	{attribute 'OPC.UA.DA' := '1'}  				                
	SP_adsorb_during_steam_bypass										: BOOL;	
	{attribute 'OPC.UA.DA' := '1'}  				                
	SP_adsorb_during_warmup												: BOOL;
	{attribute 'OPC.UA.DA' := '1'}  				                
	SP_boiler_warmup_duration											: REAL;
	{attribute 'OPC.UA.DA' := '1'}  				                
	SP_condensate_collection_tank_high_level							: REAL;	
	{attribute 'OPC.UA.DA' := '1'}  				                
	SP_condensate_collection_tank_low_level								: REAL;
	{attribute 'OPC.UA.DA' := '1'}  				                
	SP_condensation_collection_tank_emergency_low_level					: REAL;	
	{attribute 'OPC.UA.DA' := '1'}  				                
	SP_duration_to_drain_cooling_and_purge_line_in_module				: REAL;				
	{attribute 'OPC.UA.DA' := '1'}  				                
	SP_duration_to_drain_reactor_set									: REAL;	
	{attribute 'OPC.UA.DA' := '1'}  				                
	SP_evacuation_duration												: REAL;							// PS 11/25/24	
	{attribute 'OPC.UA.DA' := '1'}  				                
	SP_evacuation_ideal_pressure										: REAL;							// PS 11/25/24	
	{attribute 'OPC.UA.DA' := '1'}  				                
	SP_mass_flow_totalizer												: REAL;
	{attribute 'OPC.UA.DA' := '1'}  				                
	SP_maximum_condensate_collection_tank_refill_duration				: REAL;							// PS 08_16_24
	{attribute 'OPC.UA.DA' := '1'}  				                
	SP_maximum_condenser_knockout_drain_duration						: REAL;							// PS 08_22_24
	{attribute 'OPC.UA.DA' := '1'}  				                
	SP_maximum_duration_to_drain_reactor_set							: REAL;	
	{attribute 'OPC.UA.DA' := '1'}  				                
	SP_maximum_inlet_product_vacuum_temperature							: REAL;							// PS 04_30_24	
	{attribute 'OPC.UA.DA' := '1'}  				                
	SP_maximum_reasonable_sorbent_TC_reading							: REAL;
	{attribute 'OPC.UA.DA' := '1'}  				                
	SP_maximum_vacuum_separator_drain_duration							: REAL;							// PS 08_22_24
	{attribute 'OPC.UA.DA' := '1'}  				                
	SP_maximum_vacuum_separator_refill_duration							: REAL;							// PS 08_22_24
	{attribute 'OPC.UA.DA' := '1'}  				                
	SP_minimum_condensate_flow											: REAL;							// PS 08_22_24
	{attribute 'OPC.UA.DA' := '1'}  				                
	SP_minimum_dead_air_line_pressure									: REAL;							// PS 11/27/24
	{attribute 'OPC.UA.DA' := '1'}  				                
	SP_minimum_drainage_pressure										: REAL;	
	{attribute 'OPC.UA.DA' := '1'}  				                
	SP_minimum_reasonable_sorbent_TC_reading							: REAL;
	{attribute 'OPC.UA.DA' := '1'}  				                
	SP_minimum_steam_bypass_duration									: REAL;							// PS 12/2/24
	{attribute 'OPC.UA.DA' := '1'}  				                
	SP_minimum_steam_bypass_flow_rate									: REAL;
	{attribute 'OPC.UA.DA' := '1'}  				                
	SP_minimum_vacuum_cooling_loop_flow									: REAL := 2; 						// PS 11/25/24
	{attribute 'OPC.UA.DA' := '1'}  				                
	SP_max_vacuum_cooling_loop_temp										: REAL := 50;							// PS 11/25/24
	{attribute 'OPC.UA.DA' := '1'}  				                
	SP_minimum_vacuum_liq_seal_flow										: REAL;							// PS 08_13_24
	{attribute 'OPC.UA.DA' := '1'}  				                
	SP_product_condensate_drum_high_level								: REAL;
	{attribute 'OPC.UA.DA' := '1'}  				                
	SP_product_condensate_drum_low_level								: REAL;
	{attribute 'OPC.UA.DA' := '1'}  				                
	SP_reactor_vfd_percent_maximum										: INT;
	{attribute 'OPC.UA.DA' := '1'}  				                
	SP_reactor_vfd_percent_step_duration								: REAL;
	{attribute 'OPC.UA.DA' := '1'}  				                
	SP_reactor_vfd_percent_step_size									: INT;
	{attribute 'OPC.UA.DA' := '1'}  				                
	SP_steam_bypass_duration											: REAL;
	{attribute 'OPC.UA.DA' := '1'}  				                
	SP_steam_bypass_immediately_after_warm_up							: BOOL;
	{attribute 'OPC.UA.DA' := '1'}  				                
	SP_steam_bypass_temperature											: REAL;
	{attribute 'OPC.UA.DA' := '1'}  				                
	SP_steam_bypass_vacuum_pressure										: REAL;
	{attribute 'OPC.UA.DA' := '1'}  				                
	SP_target_boiler_pressure											: REAL;
	{attribute 'OPC.UA.DA' := '1'}  				                
	SP_vacuum_pres_control_valve										: REAL;
	{attribute 'OPC.UA.DA' := '1'}  				                
	SP_vacuum_separator_level_emergency_high							: REAL;							// PS 08_13_24									
	{attribute 'OPC.UA.DA' := '1'}  				                
	SP_vacuum_separator_level_emergency_low								: REAL;							// PS 08_13_24									
	{attribute 'OPC.UA.DA' := '1'}  				                
	SP_vacuum_separator_level_high										: REAL;							// PS 08_22_24									
	{attribute 'OPC.UA.DA' := '1'}  				                
	SP_vacuum_separator_level_mid										: REAL;							// PS 08_22_24									
	{attribute 'OPC.UA.DA' := '1'}  				                
	SP_vacuum_separator_level_low										: REAL;							// PS 08_22_24	
	{attribute 'OPC.UA.DA' := '1'}  				                
	SP_waste_water_tank_weight_full										: REAL;										
	{attribute 'OPC.UA.DA' := '1'}  				                
	SP_waste_water_tank_weight_empty									: REAL;	
	{attribute 'OPC.UA.DA' := '1'}  				                
	SP_steam_water_tank_weight_full										: REAL;										
	{attribute 'OPC.UA.DA' := '1'}  				                
	SP_steam_water_tank_weight_empty									: REAL;	
	
	
	
    /// <summary>PCV01</summary>
	vacuum_pres_control_valve_setpoint									: REAL;
	
END_VAR

// Theseus - P_U01
// Rev 1.0 - December 2, 2024

A_IO_Points();
A_PIDs();
A_MovingAverage();
A02_WarmUp();
A03_Steam_Bypass();
A08_Shutdown();
A09_Pressure_Drop_Test();
P_U01.shutdown_process													:= FALSE;

IF LEFT(gsCycleMode, 1) = '0' THEN
	IF gsCycleMode = '02' THEN
		i2Step															:= 1;
	ELSIF gsCycleMode = '03' THEN
		i3Step															:= 1;
	ELSIF gsCycleMode = '08' THEN
		i8Step															:= 1;
	ELSIF gsCycleMode = '09' THEN
		i9Step															:= 1;
	END_IF
	gsCycleMode															:= '';
END_IF

IF tonWriteData.Q OR P_U01.write_persistent_data THEN
	P_U01.write_persistent_data											:= FALSE;
	bWriteData															:= TRUE;
ELSIF NOT fbWriteData.BUSY THEN
	bWriteData															:= FALSE;
END_IF

fbWriteData(	NETID													:= '',
				PORT													:= 851,
				START													:= bWriteData,
				TMOUT													:= T#5S);

tonTimer(IN:= bTimer, PT:= REAL_TO_TIME(rTime));
tonAdsorptionTimer(IN:= bAdsorptionTimer, PT:= REAL_TO_TIME(P_M01.SP_adsorption_duration * _MINUTES));
tonWriteData(IN:= NOT bWriteData, PT:= T#30M);

// Water Scales
fb_WaterScales_In ( 
			i_value := water_scale_1 + water_scale_2,
			io_reset	:= water_scales_reset,
			o_change_value => water_scales_in_delta,
			o_change_rate => water_scales_in_rate
			);
			
fb_WaterScales_Out ( 
			i_value := water_scale_3,
			io_reset	:= water_scales_reset,
			o_change_value => water_scales_out_delta,
			o_change_rate => water_scales_out_rate
			);
		
IF water_scales_reset THEN
	water_scales_reset := FALSE;
END_IF

// Water Scales Capapcity Desorption 
condenser_tank_capacity := SP_waste_water_tank_weight_full - SP_waste_water_tank_weight_empty;
steam_delivery_tank_capacity := SP_steam_water_tank_weight_full - SP_steam_water_tank_weight_empty;
condenser_tank_room_before_full	:= SP_waste_water_tank_weight_full - water_scale_3;
steam_delivery_tank_before_empty := (water_scale_1 + water_scale_2) -  SP_steam_water_tank_weight_empty;

ACTION A_IO_Points:
// Theseus - A_IO_Points
// Rev 1.0 - November 26, 2024

interlock_condenser_steam_or_status										:= interlock_condenser_steam_or;
interlock_hot_reactor_condenser_or_status								:= interlock_hot_reactor_condenser_or;
interlock_no_steam_unevacuated_reactor_or_status						:= interlock_no_steam_unevacuated_reactor_or;
interlock_cooling_with_vacuum_or_status									:= interlock_cooling_with_vacuum_or;
interlock_separator_water_level_with_vacuum_or_status					:= interlock_separator_water_level_with_vacuum_or;
interlock_cooling_loop_flow_with_vacuum_or_status						:= interlock_cooling_loop_flow_with_vacuum_or;
interlock_condensate_tank_level_for_steam_or_status						:= interlock_condensate_tank_level_for_steam_or;
interlock_hot_sorbent_for_repressurization_or_status					:= interlock_hot_sorbent_for_repressurization_or;
interlock_reactor_over_safe_pressure_limit_or_status					:= interlock_reactor_over_safe_pressure_limit_or;
interlock_reactor_over_safe_temperature_limit_or_status					:= interlock_reactor_over_safe_temperature_limit_or;
interlock_repressurization_valve_with_steam_or_status					:= interlock_repressurization_valve_with_steam_or;
interlock_door_open_with_steam_flow_or_status							:= interlock_door_open_with_steam_flow_or;
interlock_door_open_with_reactor_vacuum_or_status						:= interlock_door_open_with_reactor_vacuum_or;
interlock_co2_adsorption_or_status										:= interlock_co2_adsorption_or;
interlock_condensate_pump_or_status										:= interlock_condensate_pump_or;
condenser_knockout_drain_or_on_status									:= condenser_knockout_drain_or_on;
condenser_knockout_drain_or_off_status									:= condenser_knockout_drain_or_off;
vacuum_separator_drain_or_on_status										:= vacuum_separator_drain_or_on;
vacuum_separator_drain_or_off_status									:= vacuum_separator_drain_or_off;
reactor_drain_or_on_status												:= reactor_drain_or_on;
reactor_drain_or_off_status												:= reactor_drain_or_off;

// Interlock 5
cooling_with_vacuum_interlock											:= NOT vacuum_liquid_loop_fan OR NOT vacuum_liquid_pump;
bCondition1																:= NOT interlock_cooling_with_vacuum_or AND cooling_with_vacuum_interlock;

// Interlock 6
separator_water_level_with_vacuum_interlock								:= vacuum_separator_level < SP_vacuum_separator_level_emergency_low OR vacuum_separator_level > SP_vacuum_separator_level_emergency_high;
bCondition2																:= NOT interlock_separator_water_level_with_vacuum_or AND separator_water_level_with_vacuum_interlock;

// Interlock 7
cooling_loop_flow_with_vacuum_interlock									:= vacuum_pump AND vacuum_pump_water_flow < SP_minimum_vacuum_liq_seal_flow;
tonVacuumInterlock(IN:= cooling_loop_flow_with_vacuum_interlock, PT:= T#5S);
bCondition3																:= NOT interlock_cooling_loop_flow_with_vacuum_or AND tonVacuumInterlock.Q;

IF bCondition1 OR bCondition2 OR bCondition3 THEN
	vacuum_pump															:= FALSE;
END_IF
IF bCondition2 THEN
	vacuum_pump_inlet_valve												:= FALSE;
	vacuum_pump_bypass_valve											:= FALSE;
	dead_air_inlet_valve												:= FALSE;
	product_line_ambient_valve											:= INT_TO_BOOL(eAmbient);
END_IF

// Interlock 8
condensate_tank_level_for_steam_interlock								:= steam_water_tank_level < SP_condensation_collection_tank_emergency_low_level;
IF NOT interlock_condensate_tank_level_for_steam_or AND condensate_tank_level_for_steam_interlock THEN
	boiler_package														:= FALSE;
	steam_water_pump													:= FALSE;
	steam_flow_control_valve											:= _CLOSED;
END_IF

gbDrainageOn															:= (drainage_on AND NOT drainage_function_off_or) OR drainage_function_on_or;

// Interlock 9
hot_sorbent_for_repressurization_interlock								:= P_M01.rs1.sorbent_high_temp >= P_M01.SP_maximum_target_sorbent_temperature_to_repressurize;
bCondition1																:= NOT interlock_hot_sorbent_for_repressurization_or AND hot_sorbent_for_repressurization_interlock;
 
// Interlock 13
P_U01.repressurization_valve_with_steam_interlock						:= NOT P_U01.steam_flow_control_valve_closed;
bCondition2																:= NOT P_U01.interlock_repressurization_valve_with_steam_or AND P_U01.repressurization_valve_with_steam_interlock;

gbRepresValves															:= NOT bCondition1 AND NOT bCondition2;

// Vacuum Separator
IF (gbDrainageOn OR vacuum_separator_drain_or_on) AND NOT vacuum_separator_drain_or_off THEN
	// Fill
	tonVacuumSeparatorFill(IN:= tap_water_feed_valve AND NOT bVacuumSeparatorFillError, PT:= REAL_TO_TIME(SP_maximum_vacuum_separator_refill_duration * _MINUTES));
	IF tonVacuumSeparatorFill.Q THEN
		tap_water_feed_valve											:= FALSE;
		bVacuumSeparatorFillError										:= TRUE;
		P_Alarms.M_Add_Alarm(_U01, gsVacuumSeparatorFillError, gsMessageTBD);
	ELSIF vacuum_separator_level < SP_vacuum_separator_level_low  AND NOT bVacuumSeparatorFillError THEN
		tap_water_feed_valve											:= TRUE;
	ELSIF vacuum_separator_level > SP_vacuum_separator_level_mid THEN
		tap_water_feed_valve											:= FALSE;
		bVacuumSeparatorFillError										:= FALSE;
	END_IF
	// Drain
//	tonVacuumSeparatorDrain(IN:= separator_drain_valve AND NOT bVacuumSeparatorDrainError, PT:= REAL_TO_TIME(SP_maximum_vacuum_separator_drain_duration * _MINUTES));
	IF tonVacuumSeparatorFill.Q THEN
		separator_drain_valve											:= FALSE;
		vacuum_separator_drain_pump										:= FALSE;
		bVacuumSeparatorDrainError										:= TRUE;
		P_Alarms.M_Add_Alarm(_U01, gsVacuumSeparatorDrainError, gsMessageTBD);
	ELSIF vacuum_separator_level >= SP_vacuum_separator_level_high THEN
		separator_drain_valve											:= TRUE;
		vacuum_separator_drain_pump										:= TRUE;
	ELSIF vacuum_separator_level < SP_vacuum_separator_level_mid THEN
		separator_drain_valve											:= FALSE;
		vacuum_separator_drain_pump										:= FALSE;
		bVacuumSeparatorDrainError										:= FALSE;
	END_IF
END_IF
rtrigVacuumSeparator(CLK:= NOT gbDrainageOn AND NOT vacuum_separator_drain_or_on AND NOT vacuum_separator_drain_or_off);
IF rtrigVacuumSeparator.Q THEN
	tap_water_feed_valve												:= FALSE;
	separator_drain_valve												:= FALSE;
	vacuum_separator_drain_pump											:= FALSE;
END_IF

// Condenser Knockout drainage
IF (gbDrainageOn OR condenser_knockout_drain_or_on) AND NOT condenser_knockout_drain_or_off THEN
	IF gbCondenserKODrainageOn THEN
//		tonCondenserKODrain(IN:= NOT bCondenserKnockoutError AND (product_condensate_drum_lsh OR product_condensate_drum_lsl), PT:= REAL_TO_TIME(SP_maximum_condenser_knockout_drain_duration * _MINUTES));
		IF tonCondenserKODrain.Q AND P_M01.rs1.reactor_condensate_flow < SP_minimum_condensate_flow THEN
			bCondenserKnockoutError										:= TRUE;
			knockout_drain_valve										:= FALSE;
			steam_flow_control_valve									:= _CLOSED;
			P_Alarms.M_Add_Alarm(_U01, gsCondenserKODrainageError, gsMessageTBD);
		ELSIF product_condensate_drum_lsh THEN
			knockout_drain_valve										:= TRUE;
		ELSIF NOT product_condensate_drum_lsh AND NOT product_condensate_drum_lsl THEN
			knockout_drain_valve										:= FALSE;
		END_IF
	ELSE
		knockout_drain_valve											:= FALSE;
	END_IF
END_IF
rtrigKODrainValve(CLK:= NOT gbDrainageOn AND NOT condenser_knockout_drain_or_on AND NOT condenser_knockout_drain_or_off);
IF rtrigKODrainValve.Q THEN
	knockout_drain_valve												:= FALSE;
END_IF

fb_adsorp_product_wastewater
	( i_execute := condenser_knockout_drain_adsorption_on,
	  i_value := P_U01.water_scale_3,
	  i_time := 30,
	  i_threshold := 1);
	  
IF condenser_knockout_drain_adsorption_on THEN
	IF NOT fb_adsorp_product_wastewater.o_below_threshold THEN
		knockout_drain_valve											:= TRUE;
	ELSIF fb_adsorp_product_wastewater.o_below_threshold OR fb_adsorp_product_wastewater.o_timeout THEN
		knockout_drain_valve											:= FALSE;
		condenser_knockout_drain_adsorption_on 							:= FALSE;
	END_IF
END_IF


IF NOT interlock_condensate_pump_or THEN
	condensate_pump														:= knockout_drain_valve OR gbCondensateValve;
END_IF

// Interlock 2
condenser_steam_interlock												:= NOT steam_flow_control_valve_closed AND (P_M01.rs1.steam_bypass_valve_open OR P_M01.rs1.product_iso_valve_open);
IF NOT interlock_condenser_steam_or AND condenser_steam_interlock THEN
	condenser_pump														:= TRUE;
	condenser_fan														:= TRUE;
END_IF

B_01																	:= boiler_package;
boiler_package_cmd_status												:= B_01;

P_01																	:= steam_water_pump;
steam_water_pump_cmd_status												:= P_01;

P_02																	:= vacuum_pump;
vacuum_pump_cmd_status													:= P_02;

P_03																	:= condensate_pump;
condensate_pump_cmd_status												:= P_03;

P_04																	:= condenser_pump;
condenser_pump_cmd_status												:= P_04;

P_05																	:= vacuum_liquid_pump;
vacuum_liquid_pump_cmd_status											:= P_05;

P_06																	:= vacuum_separator_drain_pump;
vacuum_separator_drain_pump_cmd_status									:= P_06;

E_01																	:= condenser_fan;
condenser_fan_cmd_status												:= E_01; 

X_01																	:= vacuum_liquid_loop_fan;
vacuum_liquid_loop_fan_cmd_status										:= X_01;

product_outlet_co2														:= F_AnalogIn(AT_02, product_outlet_co2_low, product_outlet_co2_high, product_outlet_co2_min, product_outlet_co2_offset);
product_outlet_co2_error												:= AT_02_error AND NOT _ProductOutletCO2ErrorOff;
bProductOutletCo2Error													:= P_Alarms.M_Check_Error(product_outlet_co2_error, bProductOutletCo2Error, _U01, gsProductOutletCo2SensorError, gsProcessCannotRun);

product_outlet_h2o														:= F_AnalogIn(AT_03, product_outlet_h2o_low, product_outlet_h2o_high, product_outlet_h2o_min, product_outlet_h2o_offset);
product_outlet_h2o_error												:= AT_03_error AND NOT _ProductOutletH2OErrorOff;
bProductOutletH2oError													:= P_Alarms.M_Check_Error(product_outlet_h2o_error, bProductOutletH2oError, _U01, gsProductOutletH2oSensorError, gsProcessCannotRun);

product_outlet_flow														:= F_AnalogIn(FT_02, product_outlet_flow_low, product_outlet_flow_high, product_outlet_flow_min, product_outlet_flow_offset);
product_outlet_flow_error												:= product_outlet_flow_error AND NOT _ProductOutletFlowErrorOff;
bProductOutletFlowError													:= P_Alarms.M_Check_Error(product_outlet_flow_error, bProductOutletFlowError, _U01, gsProductOutletFlowSensorError, gsProcessCannotRun);

condensate_flow															:= F_AnalogIn(FT_04, condensate_flow_low, condensate_flow_high, condensate_flow_min, condensate_flow_offset);
condensate_flow_error													:= FT_04_error AND NOT _CondensateFlowErrorOff;
bCondensateFlowError													:= P_Alarms.M_Check_Error(condensate_flow_error, bCondensateFlowError, _U01, gsCondensateFlowSensorError, gsProcessCannotRun);
	
tap_water_feed_flow														:= F_AnalogIn(FT_05, tap_water_feed_flow_low, tap_water_feed_flow_high, tap_water_feed_flow_min, tap_water_feed_flow_offset);
tap_water_feed_flow_error												:= FT_05_error AND NOT _TapWaterFeedFlowErrorOff;
bWaterFeedFlowError														:= P_Alarms.M_Check_Error(tap_water_feed_flow_error, bWaterFeedFlowError, _U01, gsTapWaterFeedFlowSensorError, gsProcessCannotRun);

steam_flow																:= F_AnalogIn(FT_06, steam_flow_low, steam_flow_high, steam_flow_min, steam_flow_offset);
steam_flow_error														:= FT_06_error AND NOT _SteamFlowErrorOff;
bSteamFlowError															:= P_Alarms.M_Check_Error(steam_flow_error, bSteamFlowError, _U01, gsTapWaterFeedFlowSensorError, gsProcessCannotRun);

vacuum_pump_water_flow													:= F_AnalogIn(FT_07, vacuum_pump_water_flow_low, vacuum_pump_water_flow_high, vacuum_pump_water_flow_min, vacuum_pump_water_flow_offset);
vacuum_pump_water_flow_error											:= FT_07_error AND NOT _VacuumPumpWaterFlowErrorOff;
bVacuumPumpWaterFlowError												:= P_Alarms.M_Check_Error(vacuum_pump_water_flow_error, bVacuumPumpWaterFlowError, _U01, gsVacuumPumpWaterFlowSensorError, gsProcessCannotRun);
	
condenser_flow															:= F_AnalogIn(FT_08, condenser_flow_low, condenser_flow_high, condenser_flow_min, condenser_flow_offset);
condenser_flow_error													:= FT_08_error AND NOT _CondenserFlowErrorOff;
bCondenserFlowError														:= P_Alarms.M_Check_Error(condenser_flow_error, bCondenserFlowError, _U01, gsCondenserFlowSensorError, gsProcessCannotRun);
	
steam_water_tank_level													:= F_AnalogIn(LT_01, steam_water_tank_level_low, steam_water_tank_level_high, steam_water_tank_level_min, steam_water_tank_level_offset);
steam_water_tank_level_error											:= LT_01_error AND NOT _SteamWaterTankLevelErrorOff;
bSteamWaterTankLevelError												:= P_Alarms.M_Check_Error(steam_water_tank_level_error, bSteamWaterTankLevelError, _U01, gsSteamWaterTankLevelSensorError, gsProcessCannotRun);
	
vacuum_separator_level													:= F_AnalogIn(LT_02, vacuum_separator_level_low, vacuum_separator_level_high, vacuum_separator_level_min, vacuum_separator_level_offset);
vacuum_separator_level_error											:= LT_02_error AND NOT _VacuumSeparatorLevelErrorOff;
bVacuumSeparatorLevelError												:= P_Alarms.M_Check_Error(vacuum_separator_level_error, bVacuumSeparatorLevelError, _U01, gsVacuumSeparatorLevelSensorError, gsProcessCannotRun);
	
product_vacuum_pres														:= F_AnalogIn(PT_04, product_vacuum_pres_low, product_vacuum_pres_high, product_vacuum_pres_min, product_vacuum_pres_offset);
product_vacuum_pres_error												:= PT_04_error AND NOT _ProductVacuumPresErrorOff;
bProductVacuumPresError													:= P_Alarms.M_Check_Error(product_vacuum_pres_error, bProductVacuumPresError, _U01, gsProductVacuumPresSensorError, gsProcessCannotRun);

steam_line_pres															:= F_AnalogIn(PT_07, steam_line_pres_low, steam_line_pres_high, steam_line_pres_min, steam_line_pres_offset);
steam_line_pres_error													:= PT_07_error AND NOT _SteamLinePresErrorOff;
bSteamLinePresError														:= P_Alarms.M_Check_Error(steam_line_pres_error, bSteamLinePresError, _U01, gsSteamLinePresSensorError, gsProcessCannotRun);

flow_calibration_diff_pres												:= F_AnalogIn(PDT_04, flow_calibration_diff_pres_low, flow_calibration_diff_pres_high, flow_calibration_diff_pres_min, flow_calibration_diff_pres_offset);
flow_calibration_diff_pres_error										:= PDT_04_error AND NOT _FlowCalibrationDiffPresErrorOff;
bFlowCalibrationDiffPresError											:= P_Alarms.M_Check_Error(flow_calibration_diff_pres_error, bFlowCalibrationDiffPresError, _U01, gsFlowCalibrationDiffPresSensorError, gsProcessCannotRun);


water_scale_1															:= F_AnalogIn(WI_01, water_scale_1_low, water_scale_1_high, water_scale_1_min, water_scale_1_offset);
water_scale_1_error														:= WI_01_error AND NOT _WaterScale1ErrorOff;
bWaterScale1Error														:= P_Alarms.M_Check_Error(water_scale_1_error, bWaterScale1Error, _U01, gsWaterScale1SensorError, gsWarning); 
	
water_scale_2															:= F_AnalogIn(WI_02, water_scale_2_low, water_scale_2_high, water_scale_2_min, water_scale_2_offset);
water_scale_2_error														:= WI_02_error AND NOT _WaterScale2ErrorOff;
bWaterScale2Error														:= P_Alarms.M_Check_Error(water_scale_2_error, bWaterScale2Error, _U01, gsWaterScale1SensorError, gsWarning); 

water_scale_3															:= F_AnalogIn(WI_03, water_scale_3_low, water_scale_3_high, water_scale_3_min, water_scale_3_offset);
water_scale_3_error														:= WI_03_error AND NOT _WaterScale3ErrorOff;
bWaterScale3Error														:= P_Alarms.M_Check_Error(water_scale_3_error, bWaterScale3Error, _U01, gsWaterScale1SensorError, gsWarning);

product_temp															:= F_Temperature(TT_02, product_temp_offset);
product_temp_error														:= TT_02_error AND NOT _ProductTempErrorOff;
bProductTempError														:= P_Alarms.M_Check_Error(product_temp_error, bProductTempError, _U01, gsProductTempSensorError, gsProcessCannotRun);

product_vacuum_temp														:= F_Temperature(TT_03, product_vacuum_temp_offset);
product_vacuum_temp_error												:= TT_03_error AND NOT _ProductVacuumTempOff;
bProductVacuumTempError													:= P_Alarms.M_Check_Error(product_vacuum_temp_error, bProductVacuumTempError, _U01, gsProductVacuumTempSensorError, gsProcessCannotRun);
	
inlet_line_temp															:= F_Temperature(TT_06, inlet_line_temp_offset);
inlet_line_temp_error													:= TT_06_error AND NOT _InletLineTempErrorOff;
bInletLineTempError														:= P_Alarms.M_Check_Error(inlet_line_temp_error, bInletLineTempError, _U01, gsInletLineTempSensorError, gsProcessCannotRun);

vacuum_pump_water_temp_1												:= F_Temperature(TT_10, vacuum_pump_water_temp_1_offset);
vacuum_pump_water_temp_1_error											:= TT_10_error AND NOT _VacuumPumpWaterTemp1ErrorOff;
bVacuumPumpWaterTemp1Error												:= P_Alarms.M_Check_Error(vacuum_pump_water_temp_1_error, bVacuumPumpWaterTemp1Error, _U01, gsVacuumPumpWaterTemp1SensorError, gsProcessCannotRun);

vacuum_pump_water_temp_2												:= F_Temperature(TT_11, vacuum_pump_water_temp_2_offset);
vacuum_pump_water_temp_2_error											:= TT_11_error AND NOT _VacuumPumpWaterTemp2ErrorOff;

IF bCloseXVValves THEN
	vacuum_pump_inlet_valve												:= FALSE;
	vacuum_pump_bypass_valve											:= FALSE;
	knockout_drain_valve												:= FALSE;
	dead_air_inlet_valve												:= FALSE;
	separator_drain_valve												:= FALSE;
	bCloseXVValves														:= FALSE;
END_IF

XV_03																	:= 	vacuum_pump_inlet_valve;
vacuum_pump_inlet_valve_open_cmd_status									:= vacuum_pump_inlet_valve;
vacuum_pump_inlet_valve_clear											:= F_ValveClear(vacuum_pump_inlet_valve, vacuum_pump_inlet_valve_open, vacuum_pump_inlet_valve_closed);

XV_04																	:= vacuum_pump_bypass_valve;
vacuum_pump_bypass_valve_open_cmd_status								:= XV_04;
vacuum_pump_bypass_valve_clear											:= F_ValveClear(vacuum_pump_bypass_valve, vacuum_pump_bypass_valve_open, vacuum_pump_bypass_valve_closed);

XV_06																	:= knockout_drain_valve;
knockout_drain_valve_open_cmd_status									:= XV_06;
knockout_drain_valve_clear												:= F_ValveClear(knockout_drain_valve, knockout_drain_valve_open, knockout_drain_valve_closed);

XV_10																	:= dead_air_inlet_valve;
dead_air_inlet_valve_open_cmd_status									:= dead_air_inlet_valve;
dead_air_inlet_valve_clear												:= F_ValveClear(dead_air_inlet_valve, dead_air_inlet_valve_open, dead_air_inlet_valve_closed);

XV_11																	:= product_line_ambient_valve;
product_line_ambient_valve_cmd_status									:= XV_11;
product_line_ambient_valve_clear										:= F_ValveClear(product_line_ambient_valve, product_line_ambient_valve_ambient,product_line_ambient_valve_product);

XV_12																	:= tap_water_feed_valve;
tap_water_feed_valve_cmd_status											:= XV_12;

XV_13																	:= separator_drain_valve;
separator_drain_valve_open_cmd_status									:= XV_13;
separator_drain_valve_clear												:= F_ValveClear(separator_drain_valve, separator_drain_valve_open, separator_drain_valve_closed);

XV_14																	:= steam_water_reservoir_valve;
steam_water_reservoir_valve_cmd_status									:= XV_14;

fb_Vacuum_Pres_Control_Valve_PI(		Setpoint						:= vacuum_pres_control_valve_setpoint,
										Control							:= product_vacuum_pres,
										Error							:= vacuum_pres_control_valve_position_error,
										Reverse							:= FALSE,
										Kp								:= vacuum_pres_control_valve_kp,           
										Ki								:= vacuum_pres_control_valve_ki,           
										BaseAdjust						:= vacuum_pres_control_valve_base_adjust,  
										LoopTime						:= vacuum_pres_control_valve_loop_time,    
										IBand							:= vacuum_pres_control_valve_iband,        
										Base							:= vacuum_pres_control_valve_base,         
										Mode							:= vacuum_pres_control_valve_mode,
										Input							:= vacuum_pres_control_valve,
										Mode_Out						=> vacuum_pres_control_valve_current_mode, 
										Output							=> PCV_01);

vacuum_pres_control_valve_position										:= INT_TO_REAL(PCV_01_position) / _PERCENT_FACTOR; 
vacuum_pres_control_valve_open											:= vacuum_pres_control_valve_position >= _VALVE_OPEN;
vacuum_pres_control_valve_closed										:= vacuum_pres_control_valve_position < _VALVE_CLOSED;

fb_Steam_Flow_Control_Valve_PI(			Setpoint						:= steam_flow_control_valve_setpoint,
										Control							:= ,
										Error							:= steam_flow_control_valve_position_error,
										Reverse							:= FALSE,
										Kp								:= steam_flow_control_valve_kp,           
										Ki								:= steam_flow_control_valve_ki,           
										BaseAdjust						:= steam_flow_control_valve_base_adjust,  
										LoopTime						:= steam_flow_control_valve_loop_time,    
										IBand							:= steam_flow_control_valve_iband,        
										Base							:= steam_flow_control_valve_base,         
										Mode							:= steam_flow_control_valve_mode,
										Input							:= steam_flow_control_valve,
										Mode_Out						=> steam_flow_control_valve_current_mode, 
										Output							=> PCV_02);

steam_flow_control_valve_position										:= INT_TO_REAL(PCV_02_position) / _PERCENT_FACTOR; 
steam_flow_control_valve_open											:= steam_flow_control_valve_position >= _VALVE_OPEN;
steam_flow_control_valve_closed											:= steam_flow_control_valve_position < _VALVE_CLOSED;

// ignore if < 2 Amps
l1_current_240															:= SEL(IT1 > _CURRENT_240_FACTOR * 2,0,F_IEConvert(IT1, _CURRENT_240_FACTOR));
l2_current_240															:= SEL(IT2 > _CURRENT_240_FACTOR * 2,0,F_IEConvert(IT2, _CURRENT_240_FACTOR));
l3_current_240															:= SEL(IT3 > _CURRENT_240_FACTOR * 2,0,F_IEConvert(IT3, _CURRENT_240_FACTOR));
l1_voltage_240															:= F_IEConvert(VT1, _VOLTAGE_240_FACTOR);
l2_voltage_240															:= F_IEConvert(VT2, _VOLTAGE_240_FACTOR);
l3_voltage_240															:= F_IEConvert(VT3, _VOLTAGE_240_FACTOR);

// Ignore if < 1 Amp
l1_current_120															:= SEL(IT4 > _CURRENT_120_FACTOR ,0,F_IEConvert(IT4, _CURRENT_120_FACTOR));
l1_voltage_120															:= F_IEConvert(VT4, _VOLTAGE_120_FACTOR);

// Boiler - ignore noise if < 5A = 400 counts

l1_current_boiler := SEL(IT_boiler_01 > 400, 0, F_IEConvert(IT_boiler_01, _CURRENT_BOILER_FACTOR));  // double coiled 
l2_current_boiler := SEL(IT_boiler_02 > 400, 0, F_IEConvert(IT_boiler_02, _CURRENT_BOILER_FACTOR));  // double coiled 
l3_current_boiler := SEL(IT_boiler_03 > 400, 0, F_IEConvert(IT_boiler_03, _CURRENT_BOILER_FACTOR));  // double coiled 

//boiler_ready														:= NOT boiler_outlet_pres_error AND boiler_outlet_pres > SP_target_boiler_pressure AND boiler_package;
//boiler_ready															:= boiler_ready;

tonBoilerCheck(IN:= warmup_complete AND NOT boiler_ready, PT:= _TIMEOUT_WARMUP_RESET);
IF tonBoilerCheck.Q THEN
	warmup_complete														:= FALSE;
END_IF

// These Utility errors prevent any new automated cycles from running
utility_error		:= '';
//utility_error															:= SEL(NOT boiler_ready, '', gsBoilerError);
utility_error															:= SEL(bProductVacuumPresError, utility_error, gsProductVacuumPresSensorError);
//utility_error															:= SEL(bProductOutletCo2Error, utility_error, gsProductOutletCo2SensorError);
//utility_error															:= SEL(bInletLineTempError, utility_error, gsInletLineTempSensorError);
//utility_error															:= SEL(bSteamWaterTankLevelError, utility_error, gsSteamWaterTankLevelSensorError);
utility_error															:= SEL(bVacuumSeparatorLevelError, utility_error, gsVacuumSeparatorLevelSensorError);
utility_error															:= SEL(bVacuumPumpWaterFlowError, utility_error, gsVacuumPumpWaterFlowSensorError);
utility_error															:= SEL(bVacuumPumpWaterTemp1Error, utility_error, gsVacuumPumpWaterTemp1SensorError);
//utility_error															:= SEL(bFlowCalibrationDiffPresError, utility_error, gsFlowCalibrationDiffPresSensorError);
//utility_error															:= SEL(bProductOutletH2oError, utility_error, gsProductOutletH2oSensorError);
//utility_error															:= SEL(bProductTempError, utility_error, gsProductTempSensorError);
//utility_error															:= SEL(bProductVacuumTempError, utility_error, gsProductVacuumTempSensorError);
//utility_error															:= '';

//sUtilityError															:= utility_error; // - TO BE ENABLED
END_ACTION

ACTION A_MovingAverage:
(*
moving_avg_params.nSamplesToFilter := 2;
moving_avg_params.tCtrlCycleTime := T#1000MS;
moving_avg_params.tTaskCycleTime := T#10MS;
moving_avg_params.pWorkArray_ADR := ADR(moving_avg_array);
moving_avg_params.nWorkArray_SIZEOF := SIZEOF(moving_avg_array);

moving_avg_in_sim_timer ( IN := NOT moving_avg_in_sim_timer.Q, PT := T#1000MS);

IF moving_avg_in_sim_timer.Q THEN 
	moving_avg_in := moving_avg_in + 1;
	IF moving_avg_in = 100 THEN
		moving_avg_in := 0;
	END_IF
END_IF

fb_MovingAverage(
	fIn:= moving_avg_in , 
	fManSyncValue:= , 
	bSync:= , 
	eMode:= E_CTRL_MODE.eCTRL_MODE_ACTIVE, 
	bHold:= , 
	fOut=> moving_avg_out, 
	eState=> , 
	eErrorId=> , 
	bError=> , 
	stParams:= moving_avg_params);
*)

fbMovingAverage(
	i_number_of_samples := 5,
	i_sample_time := 1000);
END_ACTION

ACTION A_PIDs:
// Steam valve

steam_valve_pid_params.tCtrlCycleTime := T#1000MS;
steam_valve_pid_params.tTaskCycleTime := T#10MS;
steam_valve_pid_params.fKp := steam_valve_pid_kp ;
steam_valve_pid_params.tTn := steam_valve_pid_tn;
steam_valve_pid_params.tTv := steam_valve_pid_tv;
steam_valve_pid_params.tTd := T#0MS;
steam_valve_pid_params.fOutMaxLimit := 100;
steam_valve_pid_params.fOutMinLimit := 0;

steam_valve_pid(
	fSetpointValue	:= steam_valve_pid_sp_value, 
	fActualValue	:= steam_valve_pid_actual_value, 
	fManSyncValue	:= steam_valve_pid_manual_sp, 
	bSync			:= FALSE, 
	eMode			:= steam_valve_pid_mode , 
	bHold:= , 
	fOut			=> steam_valve_pid_out , 
	bARWactive=> , 
	eState=> , 
	eErrorId=> , 
	bError=> , 
	stParams		:= steam_valve_pid_params);


steam_valve_pid_simulate_timer( IN := NOT steam_valve_pid_simulate_timer.Q, PT := T#10MS);
IF steam_valve_pid_simulate_timer.Q AND steam_valve_pid.eMode = E_CTRL_MODE.eCTRL_MODE_ACTIVE THEN
	//steam_valve_pid_actual_value := steam_valve_pid_actual_value * 0.8 + steam_valve_pid_out * 0.01;
	//steam_valve_pid_actual_value := steam_valve_pid_actual_value + ((steam_valve_pid_sp_value - steam_valve_pid_actual_value)/1.2) + 0.1; 
	steam_valve_pid_actual_value := steam_valve_pid_actual_value * 0.995 + steam_valve_pid_out * 0.01;
END_IF
(*	
IF steam_valve_pid.eMode = E_CTRL_MODE.eCTRL_MODE_MANUAL  AND (steam_valve_pid_sp_value <= 0) THEN
	steam_valve_pid_sp_value := steam_valve_pid_actual_value;
END_IF

IF steam_valve_pid.eMode = E_CTRL_MODE.eCTRL_MODE_ACTIVE AND (steam_valve_pid_manual_sp <= 0) THEN
	steam_valve_pid_manual_sp := steam_valve_pid_out;
END_IF
*)
simulate_process_params.tCtrlCycleTime := T#100MS;
simulate_process_params.tTaskCycleTime := T#10MS;
simulate_process_params.fKp := simulate_process_kp;
simulate_process_params.fTheta := simulate_process_dumping_ration;
simulate_process_params.tT0 := TO_TIME(simulate_process_tT0);

simulate_process(
	fIn:= steam_valve_pid_out , 
	fManValue:= , 
	eMode:= E_CTRL_MODE.eCTRL_MODE_ACTIVE, 
	bHold:= , 
//	fOut=> steam_valve_pid_actual_value , 
	eState=> , 
	eErrorId=> , 
	bError=> , 
	stParams:= simulate_process_params);
END_ACTION

ACTION A02_WarmUp:
// Theseus - P_U01.A02_WarmUp
// Rev 1.0 - October 8, 2024

CASE i2Step OF

	0:	;
		
	1:	
		sError															:= '';
		bComplete														:= FALSE;
		bRunSteamBypass													:= FALSE;
		P_U01.steam_bypass_complete										:= FALSE;
		IF NOT P_U01.warmup_complete THEN
			gsCycleStage												:= 'warm_up.initialize';							// 3
			IF NOT TRUE THEN //P_U01.boiler_outlet_pres_error THEN
				sError													:= F_Concat3(_U01, gsCycleStage, gsBoilerError);
				i2Step													:= 80;
			ELSE
				i2Step													:= i2Step + 1;
			END_IF
		ELSE
			bComplete													:= TRUE;
			i2Step														:= 90;
		END_IF
		
	2:	
		P_U01.boiler_package												:= TRUE;											// 4
		gsCycleStage													:= 'warm_up.boiler_heating';						// 5
		P_U01.drainage_on													:= TRUE;											// 6
		bAdsorptionActive												:= FALSE;											// 7
		bAdsorptionTimer												:= FALSE;
		i2Step															:= SEL(P_U01.SP_adsorb_during_warmup, 20, i2Step + 1);	// 8

	3:
		iAxStep															:= 1;												// 8.a
		i2Step															:= i2Step + 1;

	4:	
		Ax_Process_Pre_Check();																								// 8.a																			
		IF bPreCheckDone THEN
			IF sError = '' THEN																								// 8.a.i
				P_M01.rs1.repres_valves									:= P_M01.bRS01;										// 8.b
				rTime													:= _VALVE_TIME;
				i2Step													:= i2Step + 1;
			ELSE
				P_Alarms.M_Add_Alarm(CONCAT(_U01, gsCycleStage), sError, gsWarmupWillContinueWOAdsorption);					// 8.a.ii
				i2Step													:= 20;
			END_IF
		END_IF
		
	5:
		bTimer															:= TRUE;
		bPass1															:= (P_M01.bRS01 AND P_M01.rs1.repres_valves_clear) OR NOT P_M01.bRS01;
		IF bPass1 THEN
			bTimer														:= FALSE;
			i2Step														:= i2Step + 1;
		ELSIF tonTimer.Q THEN
			bTimer														:= FALSE;
			//P_M01_RS01.close_repres_valves								:= TRUE;
			//i2Step														:= 20;
			i2Step														:= i2Step + 1; 
		END_IF
		
	6:
		P_M01.rs1.open_doors											:= P_M01.bRS01;										// 8.c
		rTime															:= P_M01.SP_doorsopenclose_timedelay * _MINUTES;	// 8.c.i
		gsCycleStage													:= 'warm_up.boiler_heating_open_doors';				// 8.c.ii
		i2Step															:= i2Step + 1;

	7:
		bTimer															:= TRUE; 
		bPass1															:= (P_M01.bRS01 AND P_M01.rs1.open_doors) OR NOT P_M01.bRS01;
		IF bPass1 THEN
			bTimer														:= FALSE;
			i2Step														:= i2Step + 1;
		ELSIF tonTimer.Q THEN
			bTimer														:= FALSE;
			sRS															:= _RS01;
			P_Alarms.M_Add_Alarm(F_Concat3(_U01, sRS, gsCycleStage), gsReactorDoorOpeningError, gsWarmupWillContinueWOAdsorption);
			i2Step														:= 20;
		END_IF

	8:
		P_M01.rs1.fan_setpoint											:= SEL(P_M01.bRS01, 0, P_M01.SP_reactor_set_1_vfd_percent);	// 8.d
		gsCycleStage													:= 'warm_up.boiler_heating_turn_on_fans';			// 8.d.i
		rTime															:= _FAN_RS_DELAY_TIME;
		i2Step															:= i2Step + 1;

	9:
		bTimer															:= TRUE;
		IF tonTimer.Q THEN
			bTimer														:= FALSE;
			i2Step														:= i2Step + 1;
		END_IF

	10:
		P_M01.rs1.r1.inlet_co2_sol										:= P_M01.bRS01;										// 8.e
		P_M01.rs1.r1.outlet_co2_sol										:= P_M01.bRS01;										// 8.e
		gsCycleStage													:= 'warm_up.boiler_heating_adsorption';				// 8.e.i
		bAdsorptionTimer												:= TRUE;											// 8.f
		bAdsorptionActive												:= TRUE;											// 8.g
		i2Step															:= 20;


//**** Complete Warmup		
	20:
		P_U01.vacuum_pres_control_valve									:= _OPEN;											// 9
		rTime															:= _VALVE_TIME;
		i2Step															:= i2Step + 1;
		
	21:	
		bTimer															:= TRUE;
		IF P_U01.vacuum_pres_control_valve_open THEN																			// 9
			bTimer														:= FALSE;
			rTime														:= P_U01.SP_boiler_warmup_duration * _MINUTES;		// 11
			i2Step														:= i2Step + 1;
		ELSIF tonTimer.Q THEN
			bTimer														:= FALSE;
			sError														:= gsProductVacuumBackfeedValveError;				// 9
			IF bAdsorptionActive THEN
				P_Alarms.M_Add_Alarm(CONCAT(_U01, gsCycleStage), sError, gsProcessCannotRunAdsorptionWillContinue);
				P_U01.boiler_package										:= FALSE;
				i2Step													:= 30;
			ELSE
				i2Step													:= 80;
			END_IF
		END_IF
		
	22:
		bTimer															:= TRUE;
		IF P_U01.boiler_ready THEN																							// 12 (Handled in P_U01.A_Points)
			bTimer														:= FALSE;
			bComplete													:= TRUE;
			P_U01.warmup_complete											:= TRUE;
			i2Step														:= i2Step + 1;
		ELSIF tonTimer.Q THEN																								// 12.a
			bTimer														:= FALSE;
			sError														:= gsBoilerError;
			i2Step														:= 80;
		END_IF

	23:
		bRunSteamBypass													:= P_U01.SP_steam_bypass_immediately_after_warm_up;
		IF bAdsorptionActive AND NOT bRunSteamBypass THEN 																	// 14
			i2Step														:= 30;
		ELSIF bAdsorptionActive AND bRunSteamBypass AND NOT P_U01.SP_adsorb_during_steam_bypass THEN
			i2Step														:= 40;												// 15
		ELSE
			i2Step														:= 90;												// 13 & 16
		END_IF
	
		
//**** Adsorption 1		
	30:
		IF tonAdsorptionTimer.Q THEN																						// 14.a
			bAdsorptionTimer											:= FALSE;
			gsCycleStage												:= 'warm_up.boiler_heating.turn_off_fans';			// 14.b
			P_M01.rs1.fan_setpoint										:= 0;												// 14.c
			rTime														:= _FAN_RS_DELAY_TIME;
			i2Step														:= i2Step + 1;
		END_IF

	31:
		bTimer															:= TRUE;
		IF tonTimer.Q THEN
			bTimer														:= FALSE;
			gsCycleStage												:= 'warm_up.boiler_heating.closing_doors';			// 14.d
			P_M01.rs1.close_doors										:= TRUE;											// 14.e
			rTime														:= P_M01.SP_doorsopenclose_timedelay * _MINUTES;										// 14.e.i
			i2Step														:= i2Step + 1;
		END_IF		

	32:
		bTimer															:= TRUE;
		bPass1															:= (P_M01.bRS01 AND P_M01.rs1.inlet_doors_closed AND P_M01.rs1.outlet_doors_closed) OR NOT P_M01.bRS01;	// 14.e.ii
		IF bPass1 THEN
			bTimer														:= FALSE;
			i2Step														:= i2Step + 1;
		ELSIF tonTimer.Q THEN																								// 14.e.i
			bTimer														:= FALSE;
			bRunSteamBypass												:= FALSE;
			sRS															:= _RS01;
			P_Alarms.M_Add_Alarm(F_Concat3(_U01, sRS, gsCycleStage), gsReactorDoorClosingError, gsSystemCannotRun);
			i2Step														:= i2Step + 1;
		END_IF
		
	33:
		//P_M01_RS01.co2_sensors_on										:= FALSE;											// 14.f
		bAdsorptionActive												:= FALSE;											// 14.g
		i2Step															:= 90;

	
//**** Adsorption 2	
	40:
		IF tonAdsorptionTimer.Q THEN																						// 15.a
			bAdsorptionTimer											:= FALSE;
			P_M01.rs1.fan_setpoint										:= 0;												// 15.b
			rTime														:= _FAN_RS_DELAY_TIME;
			i2Step														:= i2Step + 1;
		END_IF

	41:
		bTimer															:= TRUE;
		IF tonTimer.Q THEN
			bTimer														:= FALSE;											// 15.c
			//P_M01_RS01.co2_sensors_on									:= FALSE;
			bAdsorptionActive											:= FALSE;											// 15.d
			i2Step														:= i2Step + 1;
		END_IF
		
	42:
		P_M01.rs1.close_doors											:= TRUE;											// 15.g
		rTime															:= P_M01.SP_doorsopenclose_timedelay * _MINUTES;										// 15.g.i
		i2Step															:= i2Step + 1;

	43:
		bTimer															:= TRUE;
		bPass1															:= (P_M01.bRS01 AND P_M01.rs1.inlet_doors_closed AND P_M01.rs1.outlet_doors_closed) OR NOT P_M01.bRS01;		// 15.g.ii
		IF bPass1 THEN
			bTimer														:= FALSE;
			i2Step														:= 90;
		ELSIF tonTimer.Q THEN
			bTimer														:= FALSE;
			bRunSteamBypass												:= FALSE;
			sRS															:= _RS01;
			P_Alarms.M_Add_Alarm(F_Concat3(_U01, sRS, gsCycleStage), gsReactorDoorOpeningError, gsSystemCannotRun);
			i2Step														:= 90;
		END_IF


//**** Process error		
	80:
		P_Alarms.M_Add_Alarm(CONCAT(_U01, gsCycleStage), sError, gsProcessCannotRun);
		gsCycleStage													:= 'warm_up.error';
		i2Step															:= i2Step + 1;

//**** Stop process		
	81:
		P_U01.vacuum_pres_control_valve									:= _CLOSED;
		//P_M01_RS01.co2_sensors_on										:= FALSE;
		P_M01.rs1.fan_setpoint											:= 0;
		rTime															:= _FAN_RS_DELAY_TIME;
		i2Step															:= i2Step + 1;

	82:
		bTimer															:= TRUE;
		IF tonTimer.Q THEN
			bTimer														:= FALSE;
			P_U01.boiler_package											:= FALSE;
			P_M01.rs1.close_doors										:= P_M01.bRS01;
			rTime														:= P_M01.SP_doorsopenclose_timedelay * _MINUTES;
			i2Step														:= 90;
		END_IF
		
//**** Close process
	90:
		gsCycleStage													:= SEL(bComplete, 'warm_up.failed', 'warm_up.complete');
		bAdsorptionTimer												:= FALSE;
		P_U01.drainage_on													:= FALSE;
		rTime															:= _PROCESS_COMPLETE_TIME;
		i2Step															:= i2Step + 1;
		
	91:
		bTimer															:= TRUE;
		IF tonTimer.Q THEN
			bTimer														:= FALSE;
			gsCycleStage												:= '';
			i2Step														:= 0;
		END_IF
				

END_CASE

IF i2Step > 0 AND i2Step < 80 AND P_U01.shutdown_process THEN
	gsCycleStage														:= 'warm_up.stopping';
	i2Step																:= 81;
END_IF
END_ACTION

ACTION A03_Steam_Bypass:
// Theseus - P_U01.A03_Steam_Bypass
// Rev 1.0 - October 7, 2024

CASE i3Step OF

	0:	;

	1:	
		bComplete														:= FALSE;
		IF P_U01.warmup_complete THEN
			IF NOT P_U01.steam_bypass_complete THEN
				gsCycleStage											:= 'steam_bypass.initialize';						// 4
				sError													:= '';
				IF P_U01.product_vacuum_pres_error THEN
					sError												:= gsProductVacuumPresSensorError;
				END_IF
				i3Step													:= SEL(sError = '', 80, i3Step + 1);
			ELSE
				bComplete												:= TRUE;
				i3Step													:= 90;
			END_IF
		ELSE
			P_U01.boiler_package										:= FALSE;
			P_Alarms.M_Add_Alarm(CONCAT(_U01, gsCycleStage), gsWarmupNotRunError, gsProcessCannotRun);
			i3Step														:= 90;
		END_IF
		
	2:	
		IF P_U01.boiler_ready THEN																							// 5.a (Handled in P_U01.A_Points)
			P_U01.bCloseXVValves										:= TRUE;											// 5.b
			rTime														:= _VALVE_TIME;
			i3Step														:= i3Step + 1;
		ELSE
			sError														:= gsBoilerError;
			sMessage													:= gsRunWarmup;
			i3Step														:= 80;
		END_IF

	3:	bTimer															:= TRUE;
		bPass1															:= P_U01.vacuum_pump_inlet_valve_closed;
		IF bPass1 THEN
			bTimer														:= FALSE;
			P_U01.vacuum_pres_control_valve								:= _OPEN;											// 5.b.iii
			rTime														:= _VALVE_TIME;
			i3Step														:= i3Step + 1;
		ELSIF tonTimer.Q THEN
			bTimer														:= FALSE;
			sError														:= SEL(bPass1, '', gsProductVacuumPumpIsoValveError);
			sError														:= SEL(bPass2, sError, gsProductVacuumOutletIsoValveError);
			i3Step														:= 80;
		END_IF
		
	4:
		bTimer															:= TRUE;
		IF P_U01.vacuum_pres_control_valve_position > _VALVE_OPEN THEN
			bTimer														:= FALSE;
			P_U01.drainage_on												:= TRUE;											// 5.c
			IF bAdsorptionActive AND P_U01.SP_adsorb_during_steam_bypass THEN													// 5.b.iv
				P_M01.rs1.open_doors									:= P_M01.bRS01;
				rTime													:= P_M01.SP_doorsopenclose_timedelay * _MINUTES;
				i3Step													:= i3Step + 1;
			ELSE
				i3Step													:= i3Step + 2;
			END_IF
		ELSIF tonTimer.Q THEN
			bTimer														:= FALSE;
			sError														:= gsProductVacuumBackfeedValveError;
			i3Step														:= 80;
		END_IF

	5:
		bTimer															:= TRUE;
		bPass1															:= (P_M01.bRS01 AND P_M01.rs1.inlet_doors_open AND P_M01.rs1.outlet_doors_open) OR NOT P_M01.bRS01;	// 5.b.iv
		IF bPass1 THEN
			bTimer														:= FALSE;
			IF NOT bAdsorptionActive AND P_U01.SP_adsorb_during_steam_bypass THEN												// 6
				iAxStep													:= 1;												// 6.b
				i3Step													:= i3Step + 1;
			ELSE
				i3Step													:= 20;
			END_IF
		ELSIF tonTimer.Q THEN
			bTimer														:= FALSE;
			bAdsorptionActive											:= FALSE;
			sRS															:= _RS01;
			P_Alarms.M_Add_Alarm(F_Concat3(_U01, sRS, gsCycleStage), gsReactorDoorOpeningError, gsSteamBypassWillContinueWOAdsorption);
			i3Step														:= 20;
		END_IF

	6:
		Ax_Process_Pre_Check();																								// 6.b																			
		IF bPreCheckDone THEN
			IF sError = '' THEN																								// 6.b.i
				P_M01.rs1.repres_valves									:= P_M01.bRS01;										// 6.c
				rTime													:= _VALVE_TIME;
				i3Step													:= i3Step + 1;
			ELSE
				P_Alarms.M_Add_Alarm(CONCAT(_U01, gsCycleStage), sError, gsSteamBypassWillContinueWOAdsorption);			// 6.b.ii
				bAdsorptionActive										:= FALSE;
				i3Step													:= 20;
			END_IF
		END_IF

	7:
		bTimer															:= TRUE;
		bPass1															:= (P_M01.bRS01 AND P_M01.rs1.repres_valves_clear) OR NOT P_M01.bRS01;
		IF bPass1 AND bPass2 AND bPass3 THEN
			bTimer														:= FALSE;
			i3Step														:= i3Step + 1;
		ELSIF tonTimer.Q THEN
			bTimer														:= FALSE;
			i3Step														:= i3Step + 1;
			//bAdsorptionActive											:= FALSE;
			//P_M01_RS01.close_repres_valves								:= P_M01.bRS01;
			//i3Step													:= 20; 
		END_IF
		
	8:
		P_M01.rs1.open_doors											:= P_M01.bRS01;
		gsCycleStage													:= 'steam_bypass.initialize.open_doors';			// 6.d.ii
		rTime															:= P_M01.SP_doorsopenclose_timedelay * _MINUTES;										// 6.d.i
		i3Step															:= i3Step + 1;

	9:
		bTimer															:= TRUE; 
		bPass1															:= (P_M01.bRS01 AND P_M01.rs1.inlet_doors_open AND P_M01.rs1.outlet_doors_open) OR NOT P_M01.bRS01;	// 6.d.ii
		IF bPass1 AND bPass2 AND bPass3 THEN
			bTimer														:= FALSE;
			i3Step														:= i3Step + 1;
		ELSIF tonTimer.Q THEN
			bTimer														:= FALSE;
			sRS															:= _RS01;
			P_Alarms.M_Add_Alarm(F_Concat3(_U01, sRS, gsCycleStage), gsReactorDoorOpeningError, gsSteamBypassWillContinueWOAdsorption);
			bAdsorptionActive											:= FALSE;
			i3Step														:= 20;
		END_IF

	10:
		P_M01.rs1.fan_setpoint											:= SEL(P_M01.bRS01, 0, P_M01.SP_reactor_set_1_vfd_percent);	// 6.e
		gsCycleStage													:= 'steam_bypass.initialize.turn_on_fans';			// 6.e.i
		rTime															:= _FAN_RS_DELAY_TIME;
		i3Step															:= i3Step + 1;

	11:
		bTimer															:= TRUE;
		IF tonTimer.Q THEN
			bTimer														:= FALSE;
			i3Step														:= i3Step + 1;
		END_IF

	12:
		//P_M01_RS01.co2_sensors_on										:= P_M01.bRS01;										// 6.f
		gsCycleStage													:= 'steam_bypass.initialize.adsorption';			// 6.f.i
		bAdsorptionTimer												:= TRUE;											// 6.a
		bAdsorptionActive												:= TRUE;											// 6.g
		i3Step															:= 20;


//**** Complete Steam Bypass		
	20:
		rSP																:= P_U01.SP_steam_bypass_vacuum_pressure;				// 8
		bPass1															:= P_U01.product_vacuum_pres < rSP;
		bPass2															:= P_U01.product_vacuum_pres < rSP;
		i3Step															:= SEL(bPass1 AND bPass2, i3Step + 1, 30);
	
	21:
		P_U01.vacuum_pump_inlet_valve										:= TRUE;											// 9.a
		rTime															:= _VALVE_TIME;
		i3Step															:= i3Step + 1;
		
	22:
		bTimer															:= TRUE;
		bPass1															:= P_U01.vacuum_pump_inlet_valve_open;
		IF bPass1 AND bPass2 THEN
			bTimer														:= FALSE;
			//P_U01.fan											:= TRUE;											// 9.a
			P_U01.vacuum_pres_control_valve								:= _CLOSED;
			i3Step														:= i3Step + 1;
		ELSIF tonTimer.Q THEN
			bTimer														:= FALSE;
			sError														:= SEL(bPass1, '', gsProductVacuumPumpIsoValveError);
			sError														:= SEL(bPass2, sError, gsProductVacuumOutletIsoValveError);
			i3Step														:= 80;
		END_IF
		
	23:	
		gsCycleStage													:= SEL(bAdsorptionActive, 'steam_bypass.evacuate_lines', 'steam_bypass.evacuate_lines.adsorption');		// 9.b.i
		rTime															:= P_M01.SP_evacuation_duration * _MINUTES;
		i3Step															:= i3Step + 1;
		
	24:
		bTimer															:= TRUE;											// 9.d
		rSP																:= P_U01.SP_steam_bypass_vacuum_pressure;
		bPass1															:= P_U01.product_vacuum_pres < rSP;
		bPass2															:= P_U01.product_vacuum_pres < rSP;
		IF bPass1 AND bPass2 THEN
			bTimer														:= FALSE;
			i3Step														:= i3Step + 1;
		ELSIF tonTimer.Q THEN
			bTimer														:= FALSE;
			sError														:= gsUnableToEvacuateLinesError;
			i3Step														:= 80;
		END_IF
	
	25:	
		P_U01.vacuum_pump_inlet_valve										:= FALSE;											// 9.e
		P_U01.vacuum_pres_control_valve									:= _OPEN;
		//P_U01.fan											:= FALSE;
		i3Step															:= 30;

		
//**** Steam Bypass		
	30:
		//P_U01.steam_bypass_valve											:= TRUE;											// 10
		gsCycleStage													:= SEL(bAdsorptionActive, 'steam_bypass.steam_bypass.adsorption', 'steam_bypass.steam_bypass');		// 10.a
		rSP																:= P_U01.SP_steam_bypass_duration * _MINUTES;				
		rTime															:= rSP;
		i3Step															:= i3Step + 1;				

	31:
		i3Step															:= i3Step + 1;
		
	32:
		P_U01.vacuum_pump_bypass_valve									:= TRUE;											// 12
		//P_U01.fan												:= TRUE;
		i3Step															:= i3Step + 1;
		
	33:
		IF TIME_TO_REAL(tonTimer.ET) >= (rSP * 0.3) THEN																	// 13
			i3Step														:= i3Step + 1;
		END_IF 
	
	34:
		i3Step															:= i3Step + 1;										// 13.a
	
	35:
		IF tonTimer.Q THEN //OR P_U01.product_line_temp > P_U01.SP_steam_bypass_temperature THEN										// 14
			bTimer														:= FALSE;
			//P_U01.steam_bypass_valve										:= FALSE;											// 15
			gsCycleStage												:= SEL(bAdsorptionActive, 'steam_bypass.wrap_up', 'steam_bypass.wrap_up.adsorption');	// 15.a
			P_U01.vacuum_pump_bypass_valve								:= FALSE;
			//P_U01.fan											:= FALSE;
			IF bAdsorptionActive THEN
				i3Step													:= 40;
			ELSE
				P_U01.steam_bypass_complete								:= TRUE;
				i3Step													:= 90;
			END_IF
		END_IF
		
		
//**** Complete Adsorption		
	40:
		IF tonAdsorptionTimer.Q THEN																						// 17.a.i
			bAdsorptionTimer											:= FALSE;
			P_M01.rs1.fan_setpoint										:= 0;												// 17.a.ii
			gsCycleStage												:= 'steam_bypass.wrap_up.turn_off_fans';			// 17.a.ii.1
			rTime														:= _FAN_RS_DELAY_TIME;
			i3Step														:= i3Step + 1;
		END_IF

	41:
		bTimer															:= TRUE;
		IF tonTimer.Q THEN
			bTimer														:= FALSE;
			P_M01.rs1.close_doors										:= TRUE;											// 17.a.iii
			gsCycleStage												:= 'steam_bypass.wrap_up.close_doors';				// 17.a.iii.1
			rTime														:= P_M01.SP_doorsopenclose_timedelay * _MINUTES;										// 17.a.iii.2
			i3Step														:= i3Step + 1;
		END_IF		

	42:
		bTimer															:= TRUE;
		bPass1															:= (P_M01.bRS01 AND P_M01.rs1.inlet_doors_closed AND P_M01.rs1.outlet_doors_closed) OR NOT P_M01.bRS01;		// 17.a.iii.3
		IF bPass1 AND bPass2 AND bPass3 THEN
			bTimer														:= FALSE;
			i3Step														:= i3Step + 1;
		ELSIF tonTimer.Q THEN
			bTimer														:= FALSE;
			sRS															:= _RS01;
			P_Alarms.M_Add_Alarm(F_Concat3(_U01, sRS, gsCycleStage), gsReactorDoorClosingError, gsSystemCannotRun);
			i3Step														:= i3Step + 1;
		END_IF
		
	43:
		//P_M01_RS01.co2_sensors_on										:= FALSE;											// 17.a.iv
		bAdsorptionActive												:= FALSE;											// 17.a.v
		i3Step															:= 90;

	
//**** Process error		
	80:
		gsCycleStage													:= 'steam_bypass.error';
		sMessage														:= SEL(sMessage = gsRunWarmup, gsProcessCannotRun, sMessage);
		P_Alarms.M_Add_Alarm(CONCAT(_U01, gsCycleStage), sError, sMessage);
		i3Step															:= i3Step + 1;

//**** Stop process
	81:
		//P_M01_RS01.co2_sensors_on										:= FALSE;
		P_M01.rs1.fan_setpoint											:= 0;
		rTime															:= _FAN_RS_DELAY_TIME;
		i3Step															:= i3Step + 1;

	82:
		bTimer															:= TRUE;
		IF tonTimer.Q THEN
			bTimer														:= FALSE;
			i3Step														:= i3Step + 1;
		END_IF

	83:
		//P_U01.fan												:= FALSE;
		P_U01.vacuum_pump_bypass_valve									:= FALSE;
		P_U01.vacuum_pres_control_valve									:= _CLOSED;
		P_U01.vacuum_pump_inlet_valve									:= FALSE;
		rTime															:= _VALVE_TIME;
		i3Step															:= i3Step + 1;
		
	84:
		bTimer															:= TRUE;
		IF tonTimer.Q THEN
			bTimer														:= FALSE;
			i3Step														:= 90;
		END_IF
		
//**** Close process
	90:
		gsCycleStage													:= SEL(bComplete, 'steam_bypass.failed', 'steam_bypass.complete');
		bAdsorptionTimer												:= FALSE;
		P_U01.drainage_on												:= FALSE;
		rTime															:= _PROCESS_COMPLETE_TIME;
		i3Step															:= i3Step + 1;
		
	91:
		bTimer															:= TRUE;
		IF tonTimer.Q THEN
			bTimer														:= FALSE;
			gsCycleStage												:= '';
			i3Step														:= 0;
		END_IF
				
END_CASE

IF i3Step > 0 AND i3Step < 80 AND P_U01.shutdown_process THEN
	gsCycleStage														:= 'steam_bypass.stopping';
	i3Step																:= 81;
END_IF
END_ACTION

ACTION A08_Shutdown:
// Theseus - P_U01.A08_Shutdown
// Rev 1.0 - October 7, 2024

CASE i8Step OF

	0:	;

	1:	
		bComplete														:= FALSE;
		gsCycleStage													:= 'shutdown.initialize';							// 1.a
		P_U01.boiler_package												:= FALSE;											// 3
		i8Step															:= i8Step + 1;

	2:
		P_M01.rs1.fan_setpoint											:= 0;
		rTime															:= _PAUSE_TIME;
		i8Step															:= i8Step + 1;
		
	3:
		bTimer															:= TRUE;
		IF tonTimer.Q THEN
			bTimer														:= FALSE;						
			P_M01.rs1.close_doors										:= P_M01.bRS01;										// 4
			gsCycleStage												:= 'shutdown.close_doors';							// 4.a
			rTime														:= P_M01.SP_doorsopenclose_timedelay * _MINUTES;
			i8Step														:= i8Step + 1;
		END_IF

	4:
		bTimer															:= TRUE; 
		bPass1															:= (P_M01.bRS01 AND P_M01.rs1.inlet_doors_closed AND P_M01.rs1.outlet_doors_closed) OR NOT P_M01.bRS01;
		IF bPass1 OR tonTimer.Q THEN
			IF tonTimer.Q THEN 
				sRS														:= _RS01;
				P_Alarms.M_Add_Alarm(F_Concat3(_U01, gsCycleStage, sRS), gsReactorDoorClosingError, gsSystemCannotRun);
			END_IF
			bTimer														:= FALSE;
			i8Step														:= i8Step + 1;
		END_IF

	5:
		P_M01.rs1.close_valves											:= P_M01.bRS01;										// 5		
		gsCycleStage													:= 'shutdown.wrap_up';								// 5.a
		rTime															:= _VALVE_TIME;
		i8Step															:= i8Step + 1;
		
	6:
		bTimer															:= TRUE;
		IF tonTimer.Q THEN
			bTimer														:= FALSE;
			//P_M01_RS01.co2_sensors_on									:= NOT P_M01.bRS01;
			P_M01.rs1.repres_valves										:= NOT P_M01.bRS01;
			i8Step														:= i8Step + 1;
		END_IF
		
	7:
		P_U01.bCloseXVValves											:= TRUE;
		P_U01.vacuum_pres_control_valve									:= 0;
		rTime															:= _PAUSE_TIME;
		i8Step															:= i8Step + 1;

	8:
		bTimer															:= TRUE;
		bPass1															:= NOT P_M01.rs1.reactor_drain_vessel_lsl;			// 6
		bPass2															:= NOT product_condensate_drum_lsh;
		gsCycleStage													:= 'shutdown.drain';								// 6.a
		IF bPass1 AND bPass2 THEN
			bTimer														:= FALSE;
 		ELSIF tonTimer.Q THEN
			sError														:= SEL(NOT bPass1, '', F_concat3(_RS01, ' ', gsCondensateLslError));
			sError														:= SEL(NOT bPass2, sError, gsProductCondensateDrumLshError);
			P_Alarms.M_Add_Alarm(_U01, sError, gsCheckOperation);
		END_IF
		i8Step															:= 90;
		
//**** Close process
	90:
		gsCycleStage													:= 'shutdown.complete';								// 7
		rTime															:= _PROCESS_COMPLETE_TIME;
		i8Step															:= i8Step + 1;
		
	91:
		bTimer															:= TRUE;
		IF tonTimer.Q THEN
			bTimer														:= FALSE;
			gsCycleStage												:= '';
			i8Step														:= 0;
		END_IF
				
END_CASE

IF i8Step > 0 AND i8Step < 80 AND P_U01.shutdown_process THEN
	gsCycleStage														:= 'shutdown.stopping';
	i8Step																:= 81;
END_IF
END_ACTION

ACTION A09_Pressure_Drop_Test:
// Theseus - P_U01.A09_Pressure_Drop_Test
// Rev 1.0 - October 8, 2024

CASE i9Step OF

	0:	;

	1:	
		bComplete														:= FALSE;
		gsCycleStage													:= 'pressure_drop_test.initialize';					// 3
		i9Step															:= i9Step + 1;

	2:	
		Ax_Process_Pre_Check();																								// 3.a																			
		IF bPreCheckDone THEN
			IF sError = '' THEN																								// 3.a.i
				P_U01.drainage_on											:= TRUE;											// 3.c
				i9Step													:= i9Step + 1;
			ELSE
				sRS														:= '';
				sMessage												:= gsPressureDropTestCannotRun;						// 3.a.ii
				i9Step													:= 80;
			END_IF
		END_IF

	3:
		P_M01.rs1.repres_valves											:= P_M01.bRS01;										// 4
		rTime															:= _VALVE_TIME;
		i9Step															:= i9Step + 1;

	4:
		bTimer															:= TRUE;
		bPass1															:= (P_M01.bRS01 AND P_M01.rs1.repres_valves_clear) OR NOT P_M01.bRS01;
		IF bPass1 OR tonTimer.Q THEN
			bTimer														:= FALSE;
			i9Step														:= i9Step + 1;
		END_IF
		
	5:
		P_M01.rs1.open_doors											:= P_M01.bRS01;										// 5
		gsCycleStage													:= 'pressure_drop_test.open_doors';					// 5.a
		rTime															:= P_M01.SP_doorsopenclose_timedelay * _MINUTES;		// 5.b
		i9Step															:= i9Step + 1;

	6:
		bTimer															:= TRUE; 
		bPass1															:= (P_M01.bRS01 AND P_M01.rs1.inlet_doors_open AND P_M01.rs1.outlet_doors_open) OR NOT P_M01.bRS01;	// 5.c
		IF bPass1 THEN
			bTimer														:= FALSE;
			iVfd_Speed													:= P_U01.SP_reactor_vfd_percent_step_size;			// 6
			bVfd_Speed_Up												:= TRUE;
			gsCycleStage												:= 'pressure_drop_test.pressure_drop_test';			// 6.a
			rTime														:= P_U01.SP_reactor_vfd_percent_step_duration * _MINUTES;	// 7
			i9Step														:= i9Step + 1;
		ELSIF tonTimer.Q THEN
			bTimer														:= FALSE;
			sRS															:= _RS01;
			sError														:= gsReactorDoorOpeningError;
			sMessage													:= gsPressureDropTestCannotRun;
			i9Step														:= 80;
		END_IF

	7:
		P_M01.rs1.fan_setpoint											:= SEL(P_M01.bRS01, 0, iVfd_Speed);
		i9Step															:= SEL(iVfd_Speed = 0, i9Step + 1, i9Step + 2);		//11

	8:
		bTimer															:= TRUE;
		IF tonTimer.Q THEN																									// 8
			bTimer														:= FALSE;
			IF bVfd_Speed_Up THEN
				IF iVfd_Speed + P_U01.SP_reactor_vfd_percent_step_size <= P_U01.SP_reactor_vfd_percent_maximum THEN
					iVfd_Speed											:= iVfd_Speed + P_U01.SP_reactor_vfd_percent_step_size;	// 9
				ELSE
					bVfd_Speed_Up										:= FALSE;
					iVfd_Speed											:= iVfd_Speed - P_U01.SP_reactor_vfd_percent_step_size;
				END_IF
			ELSE
				IF iVfd_Speed - P_U01.SP_reactor_vfd_percent_step_size >= 0 THEN
					iVfd_Speed											:= iVfd_Speed - P_U01.SP_reactor_vfd_percent_step_size;	// 10
				ELSE
					iVfd_Speed											:= 0;
				END_IF
			END_IF
			i9Step														:= i9Step - 1;
		END_IF

	9:
		bComplete														:= TRUE;
		gsCycleStage													:= 'pressure_drop_test.close_doors';				// 11.a
		P_M01.rs1.close_doors											:= P_M01.bRS01;										// 12
		rTime															:= P_M01.SP_doorsopenclose_timedelay * _MINUTES;										// 12.a
		i9Step															:= i9Step + 1;

	10:
		bTimer															:= TRUE;
		bPass1															:= (P_M01.bRS01 AND P_M01.rs1.inlet_doors_closed and P_M01.rs1.outlet_doors_closed) OR NOT P_M01.bRS01;	// 12.b
		IF bPass1 THEN
			bTimer														:= FALSE;
			i9Step														:= i9Step + 1;
		ELSIF tonTimer.Q THEN
			bTimer														:= FALSE;
			sRS															:= _RS01;
			P_Alarms.M_Add_Alarm(F_Concat3(_U01, gsCycleStage, sRS), gsReactorDoorClosingError, gsUnableToCloseDoors);
			i9Step														:= 90;
		END_IF
		

//**** Process error		
	80:
		gsCycleStage													:= 'pressure_drop_test.error';
		P_Alarms.M_Add_Alarm(F_Concat3(_U01, sRS, gsCycleStage), sError, sMessage);
		i9Step															:= i9Step + 1;

//**** Stop process		
	81:
		P_M01.rs1.fan_setpoint											:= 0;
		i9Step															:= 90;
		
//**** Close process
	90:
		gsCycleStage													:= SEL(bComplete, 'pressure_drop_test.failed', 'pressure_drop_test.complete');	// 13
		P_U01.drainage_on													:= FALSE;
		rTime															:= _PROCESS_COMPLETE_TIME;
		i9Step															:= i9Step + 1;
		
	91:
		bTimer															:= TRUE;
		IF tonTimer.Q THEN
			bTimer														:= FALSE;
			gsCycleStage												:= '';
			i9Step														:= 0;
		END_IF
				
END_CASE

IF i9Step > 0 AND i9Step < 80 AND P_U01.shutdown_process THEN
	gsCycleStage														:= 'pressure_drop_test.stopping';
	i9Step																:= 81;
END_IF
END_ACTION

ACTION Ax_Process_Pre_Check:
// Theseus - P_U01.Ax_Process_Pre_Check
// Rev 1.0 - October 7, 2024

CASE iAxStep OF

	0:	;

	1:	
		sError															:= '';
		bPreCheckDone													:= FALSE;
		P_M01.rs1.close_valves											:= P_M01.bRS01;
		P_M01.rs1.retract_clamps										:= P_M01.bRS01;
		rTime															:= _VALVE_TIME;
		iAxStep															:= iAxStep + 1;
	
	2:	
		bTimer															:= TRUE;
		bPass1															:= (P_M01.bRS01 AND P_M01.rs1.rs_valves_clear) OR NOT P_M01.bRS01;
		IF bPass1 THEN
			bTimer														:= FALSE;
			iAxStep														:= iAxStep + 1;
		ELSIF tonTimer.Q THEN
			sError														:= 'Valve Error';
			iAxStep														:= 99;
		END_IF

	3:
		IF P_M01.rs1.adsorption_high_temp_count <= _HIGH_CART_READINGS_MAX THEN
			iAxStep														:= iAxStep + 1;
		ELSE
			sError														:= gsHighTempCountError;
			iAxStep														:= 99;
		END_IF

	4:
		bPass1															:= (P_M01.bRS01 AND P_M01.rs1.inlet_clamps_retracted) OR NOT P_M01.bRS01; 
		IF bPass1 AND bPass2 AND bPass3 THEN
			iAxStep														:= iAxStep + 1;
		ELSE
			sError														:= gsClampRetractError;
			iAxStep														:= 99;
		END_IF
		
	5:
		iAxStep															:= iAxStep + 1;
		
	6:
		///@@@bPass1															:= (P_M01.bRS01 AND P_M01.rs1.average_pressure_within_ambient) OR NOT P_M01.bRS01;
		IF NOT bPass1 OR NOT bPass2 OR NOT bPass3 THEN
			sError														:=  gsAmbientPressureError;
		END_IF
		iAxStep															:= 99;
		
	99:
		bTimer															:= FALSE;
		bPreCheckDone													:= TRUE;
		iAxStep															:= 0;
				
END_CASE
END_ACTION

END_PROGRAM

// ---- POUs/Function_Blocks/FB_PI_Control.TcPOU
FUNCTION_BLOCK FB_PI_Control
VAR_INPUT
	Setpoint											: REAL;									// Target value
	Control												: REAL;									// Actual value
	Input												: REAL	:= 0;							// Value to set output in manual mode
	Minimum_Output										: REAL	:= 0;							// Minimum output in auto mode
	LoopTime											: REAL	:= 500;							// PI loop time in msecs
	Kp													: REAL	:= 100;							// Proportional constant
	Ki													: REAL	:= 0.05;						// Integral constant
	IBand												: REAL	:= 3;							// Plus/minus range within setpoint that Integral is active
	Base												: INT	:= 16384;						// Ideal output to hit setpoint
	BaseAdjust											: INT	:= 10;							// Amount to adjust base value if not within IBand range 
	Mode												: INT	:= 0;							// 0 = Off, 1 = Manual, 2 = Modulation, 3 = Autotune (not currently implemented)
	Error												: BOOL;
	Reverse												: BOOL;
END_VAR                                 		
VAR_OUTPUT                              		
	Output												: INT;
	Mode_Out											: INT;
END_VAR                                 		
VAR                                     		
	bNegativeError										: BOOL;
	bLastError											: BOOL;
	rError												: REAL;
	rBase												: INT;
	P													: REAL;
	I													: REAL;
	MinOut												: INT;
	tonLoop												: TON;
END_VAR

// FB_PI_Control
// Rev 1.0 - April 24, 2024

MinOut													:= REAL_TO_INT(Minimum_Output * _PERCENT_FACTOR);
IF Mode = eOff OR Mode > eAuto THEN // OR Error THEN
	Output												:= 0;
	I													:= 0;													// Reset Integral error 
	rBase												:= Base;
ELSIF Mode = eManual THEN
	Output												:= REAL_TO_INT(Input * _PERCENT_FACTOR);				// Manual
	rBase												:= Base;
ELSIF Mode = eAuto THEN																							// Modulation
	IF tonLoop.Q THEN
		tonLoop(IN:= FALSE);	
		rError											:= SEL(Reverse, Setpoint - Control, Control - Setpoint);
		bNegativeError									:= rError > 0;
		IF bNegativeError <> bLastError THEN																	// Zero crossover
			bLastError									:= bNegativeError;
			rBase										:= REAL_TO_INT(rBase + I);
			rBase										:= SEL(rBase < 0, SEL(rBase > 32767, rBase, 32767), 0);
			I											:= 0;
		END_IF
		P												:= rError * Kp;
		I												:= SEL(ABS(rError) < IBand, 0, I + (rError * Ki));
		IF ABS(rError) > IBand THEN
			rBase										:= SEL(bNegativeError, rBase - BaseAdjust, rBase + BaseAdjust);
			rBase										:= SEL(rBase < 0, SEL(rBase > 32767, rBase, 32767), 0);
		END_IF
		Output											:= REAL_TO_INT(rBase + P + I);
		Output											:= SEL(Output < MinOut, Output, MinOut);
	END_IF
	
	tonLoop(IN:= TRUE, PT:= REAL_TO_TIME(LoopTime));
ELSIF Mode = eTune THEN
	;																											// Autotune (TBC)
END_IF

Mode_Out												:= Mode;
Output													:= SEL(Output < 0, SEL(Output > 32767, Output, 32767), 0);

END_FUNCTION_BLOCK

// ---- POUs/Function_Blocks/FB_RateOfChange.TcPOU
FUNCTION_BLOCK FB_RateOfChange
VAR_INPUT
	i_value : REAL;
	io_reset : BOOL;
END_VAR
VAR_OUTPUT
	o_change_value : REAL;
	o_change_rate : REAL;
END_VAR
VAR_IN_OUT
//	io_reset : BOOL;
END_VAR
VAR
	value_reset : REAL;   // value at reset 

	tmr_Reset : TON := ( PT := T#24H);
	time_since_reset : REAL;  // seconds
END_VAR

// 600 minute timer to get the total 
tmr_Reset(IN := NOT io_reset);

time_since_reset := TO_REAL( tmr_Reset.ET) / 1000;



IF io_reset THEN
	value_reset := i_value;
	o_change_rate := 0;
	o_change_value := 0;
//	io_reset := FALSE;
ELSIF time_since_reset > 0 THEN
	o_change_value := i_value - value_reset;
	o_change_rate := o_change_value / time_since_reset;
END_IF

END_FUNCTION_BLOCK

// ---- POUs/Function_Blocks/FB_MovingAverage.TcPOU
FUNCTION_BLOCK FB_MovingAverage
VAR_INPUT
	i_value_to_avg													: REAL;
	i_number_of_samples												: UINT;
	i_sample_time													: UINT;  // ms
END_VAR
VAR_OUTPUT
	o_avg_value												: LREAL;
END_VAR
VAR
	fb_CtrlMovingAverage											: FB_CTRL_MOVING_AVERAGE;
	moving_avg_params												: ST_CTRL_MOVING_AVERAGE_PARAMS;
	moving_avg_array												: ARRAY[1..1000] OF REAL;
	moving_avg_in_sim_timer											: TON;
END_VAR

moving_avg_params.nSamplesToFilter := i_number_of_samples;
moving_avg_params.tCtrlCycleTime := TO_TIME(i_sample_time);
moving_avg_params.tTaskCycleTime := T#10MS;
moving_avg_params.pWorkArray_ADR := ADR(moving_avg_array);
moving_avg_params.nWorkArray_SIZEOF := SIZEOF(moving_avg_array);

moving_avg_in_sim_timer ( IN := NOT moving_avg_in_sim_timer.Q, PT := T#1000MS);

IF moving_avg_in_sim_timer.Q THEN 
	i_value_to_avg := i_value_to_avg + 1;
	IF i_value_to_avg = 30 THEN
		i_value_to_avg := 0;
	END_IF
END_IF

fb_CtrlMovingAverage(
	fIn:= i_value_to_avg , 
	fManSyncValue:= , 
	bSync:= , 
	eMode:= E_CTRL_MODE.eCTRL_MODE_ACTIVE, 
	bHold:= , 
	fOut=> o_avg_value, 
	eState=> , 
	eErrorId=> , 
	bError=> , 
	stParams:= moving_avg_params);

END_FUNCTION_BLOCK

// ---- POUs/Functions/F_ValveClear.TcPOU
FUNCTION F_ValveClear : bool
VAR_INPUT
	Input																: BOOL;
	Open																: BOOL;
	Closed																: BOOL;
END_VAR
VAR
END_VAR

// F_ValveClear
// Rev 1.0 - December 28, 2023

F_ValveClear															:= ((Input AND Open) OR (NOT Input AND Closed)) AND NOT (Open = Closed);

END_FUNCTION

// ---- POUs/Functions/F_IEConvert.TcPOU
FUNCTION F_IEConvert : REAL
VAR_INPUT
	Input																: INT;
	Factor																: REAL;
END_VAR
VAR
END_VAR

// F_IEConvert
// Rev 1.0 - December 28, 2023

F_IEConvert															:= INT_TO_REAL(Input) / Factor;

END_FUNCTION

// ---- POUs/Functions/F_LowMidHigh.TcPOU
/// <summary>Returns 0 if Value < Low, 2 if Value > High, 1 otherwise</summary>
FUNCTION F_LowMidHigh : INT
VAR_INPUT
	Value																: REAL;
	Low																	: REAL;
	High																: REAL;
	Current																: INT;
END_VAR
VAR
	Out																	: INT;
END_VAR

// F_LowMidHigh
// Rev 1.0 - April 19, 2024

IF Value > High THEN
	Out																	:= 2;
ELSIF Value >= Low THEN
	Out																	:= 1;
ELSE
	Out																	:= 0;
END_IF
F_LowMidHigh															:= F_HighestInt(Value1:= Out, Value2:= Current);

END_FUNCTION

// ---- POUs/Functions/F_Concat4.TcPOU
FUNCTION F_Concat4 : STRING
VAR_INPUT
	s1																	: STRING;
	s2																	: STRING;
	s3																	: STRING;
	s4																	: STRING;
END_VAR
VAR
END_VAR

// F_Concat4
// Rev 1.0 - January 10, 2024

F_Concat4																:= CONCAT(s1, s2);
F_Concat4																:= CONCAT(F_Concat4, s3);
F_Concat4																:= CONCAT(F_Concat4, s4);

END_FUNCTION

// ---- POUs/Function_Blocks/FB_Analog_Out.TcPOU
FUNCTION_BLOCK FB_Analog_Out
VAR_INPUT
END_VAR
VAR_IN_OUT
	Input1																: REAL;
	Input2																: REAL;
END_VAR
VAR
	Last1																: REAL;
	Last2																: REAL;
END_VAR

// Theseus - FB_Analog_Out
// Rev 1.0 - April 3, 2024

IF Input2 <> Last2 THEN
	Last2																:= Input2;
	Input1																:= Input2;
	Last1																:= Input2;
ELSIF Input1 <> Last1 THEN
	Last1																:= Input1;
	Input2																:= Input1;
	Last2																:= Input1;
END_IF

END_FUNCTION_BLOCK

// ---- POUs/Function_Blocks/FB_Integer_Out.TcPOU
FUNCTION_BLOCK FB_Integer_Out
VAR_INPUT
END_VAR
VAR_IN_OUT
	Input1																: INT;
	Input2																: INT;
END_VAR
VAR
	Last1																: INT;
	Last2																: INT;
END_VAR

// Theseus - FB_Integer_Out
// Rev 1.0 - April 24, 2024

IF Input2 <> Last2 THEN
	Last2																:= Input2;
	Input1																:= Input2;
	Last1																:= Input2;
ELSIF Input1 <> Last1 THEN
	Last1																:= Input1;
	Input2																:= Input1;
	Last2																:= Input1;
END_IF

END_FUNCTION_BLOCK

// ---- POUs/Function_Blocks/FB_ValveError.TcPOU
FUNCTION_BLOCK PUBLIC FB_ValveError
VAR_INPUT
	Command																: BOOL;
	Open																: BOOL;
	Closed																: BOOL;
END_VAR
VAR_OUTPUT
	ti_Status																: INT;
END_VAR
VAR
	Transition															: BOOL;
	tonError															: TON;
END_VAR

//// Theseus - FB_ValveError
//// Rev 1.0 - December 28, 2023

Transition																:= (Command AND NOT Open) OR (NOT Command AND NOT Closed);
ti_Status																	:= SEL(Transition, 0, SEL(tonError.Q, 1, 2)); 

tonError(IN:= Transition, PT:= REAL_TO_TIME(_VALVE_TIME * _SECONDS));

END_FUNCTION_BLOCK
